// Mitsubishi GX Works2 project: 158-NGUYEN VAN CU   PLC: FX3G

PROGRAM MAIN
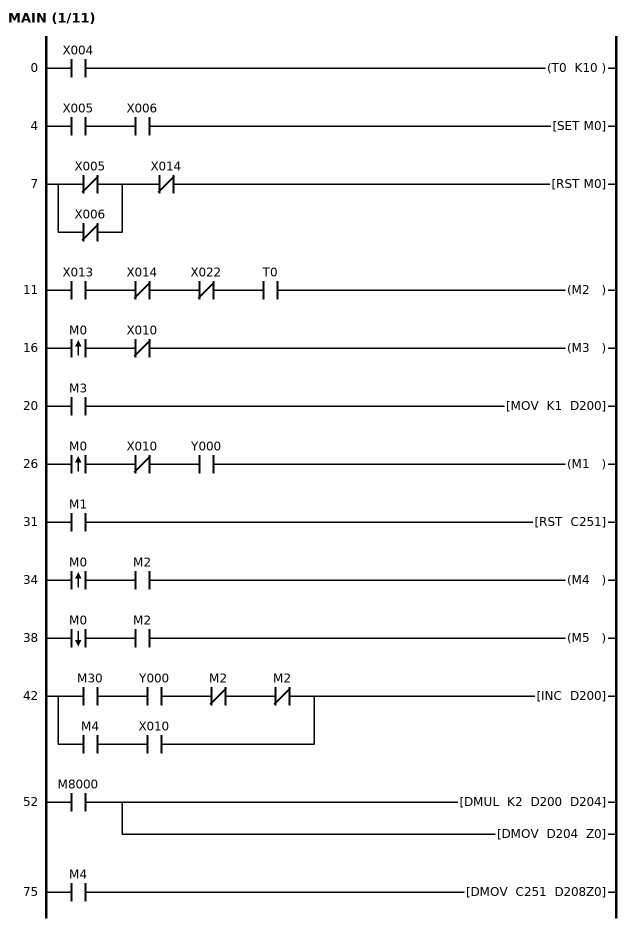
0     LD      X004
      OUT     T0 K10
4     LD      X005
      AND     X006
      SET     M0
7     LDI     X005
      ORI     X006
      ANI     X014
      RST     M0
11    LD      X013
      ANI     X014
      ANI     X022
      AND     T0
      OUT     M2
16    LDP     M0
      ANI     X010
      OUT     M3
20    LD      M3
      MOV     K1 D200
26    LDP     M0
      ANI     X010
      AND     Y000
      OUT     M1
31    LD      M1
      RST     C251
34    LDP     M0
      AND     M2
      OUT     M4
38    LDF     M0
      AND     M2
      OUT     M5
42    LD      M30
      AND     Y000
      ANI     M2
      ANI     M2
      LD      M4
      AND     X010
      ORB
      INC     D200
52    LD      M8000
      DMUL    K2 D200 D204
      DMOV    D204 Z0
75    LD      M4
      DMOV    C251 D208Z0
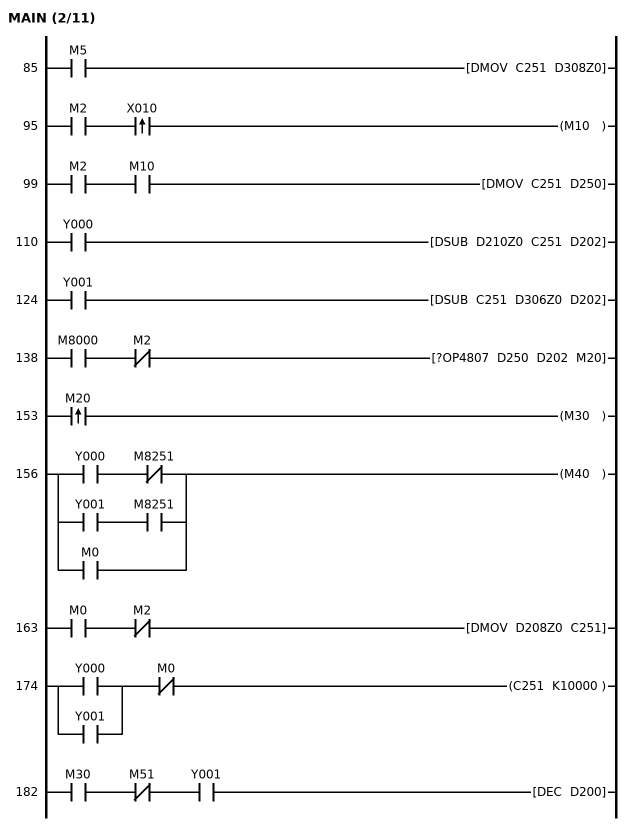
85    LD      M5
      DMOV    C251 D308Z0
95    LD      M2
      ANDP    X010
      OUT     M10
99    LD      M2
      AND     M10
      DMOV    C251 D250
110   LD      Y000
      DSUB    D210Z0 C251 D202
124   LD      Y001
      DSUB    C251 D306Z0 D202
138   LD      M8000
      ANI     M2
      ?OP4807 D250 D202 M20
153   LDP     M20
      OUT     M30
156   LD      Y000
      ANI     M8251
      LD      Y001
      AND     M8251
      ORB
      OR      M0
      OUT     M40
163   LD      M0
      ANI     M2
      DMOV    D208Z0 C251
174   LD      Y000
      OR      Y001
      ANI     M0
      OUT     C251 K10000
182   LD      M30
      ANI     M51
      AND     Y001
      DEC     D200
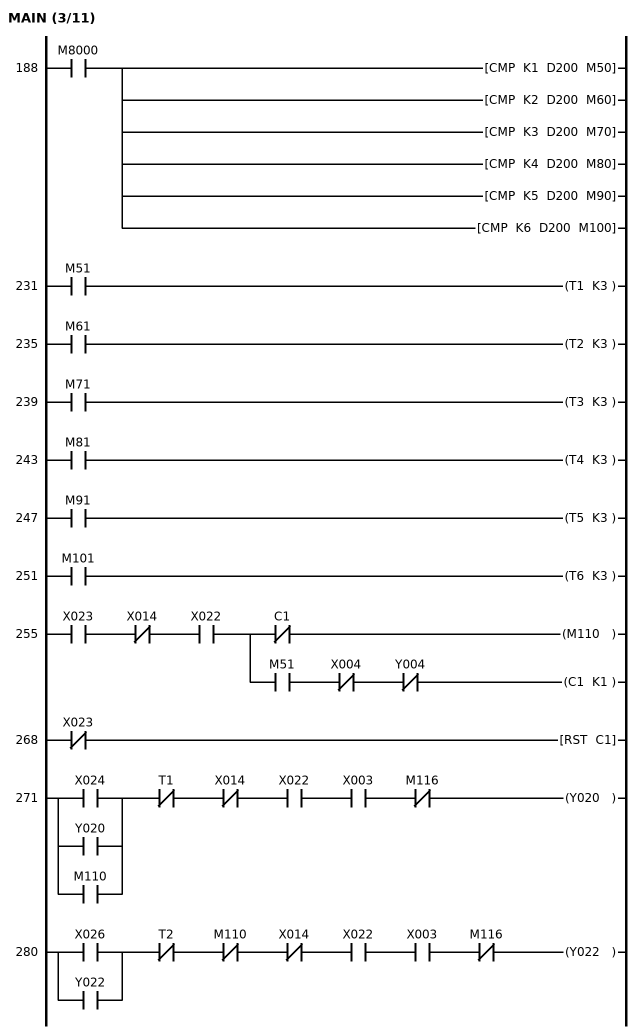
188   LD      M8000
      CMP     K1 D200 M50
      CMP     K2 D200 M60
      CMP     K3 D200 M70
      CMP     K4 D200 M80
      CMP     K5 D200 M90
      CMP     K6 D200 M100
231   LD      M51
      OUT     T1 K3
235   LD      M61
      OUT     T2 K3
239   LD      M71
      OUT     T3 K3
243   LD      M81
      OUT     T4 K3
247   LD      M91
      OUT     T5 K3
251   LD      M101
      OUT     T6 K3
255   LD      X023
      ANI     X014
      AND     X022
      MPS
      ANI     C1
      OUT     M110
      MPP
      AND     M51
      ANI     X004
      ANI     Y004
      OUT     C1 K1
268   LDI     X023
      RST     C1
271   LD      X024
      OR      Y020
      OR      M110
      ANI     T1
      ANI     X014
      AND     X022
      AND     X003
      ANI     M116
      OUT     Y020
280   LD      X026
      OR      Y022
      ANI     T2
      ANI     M110
      ANI     X014
      AND     X022
      AND     X003
      ANI     M116
      OUT     Y022
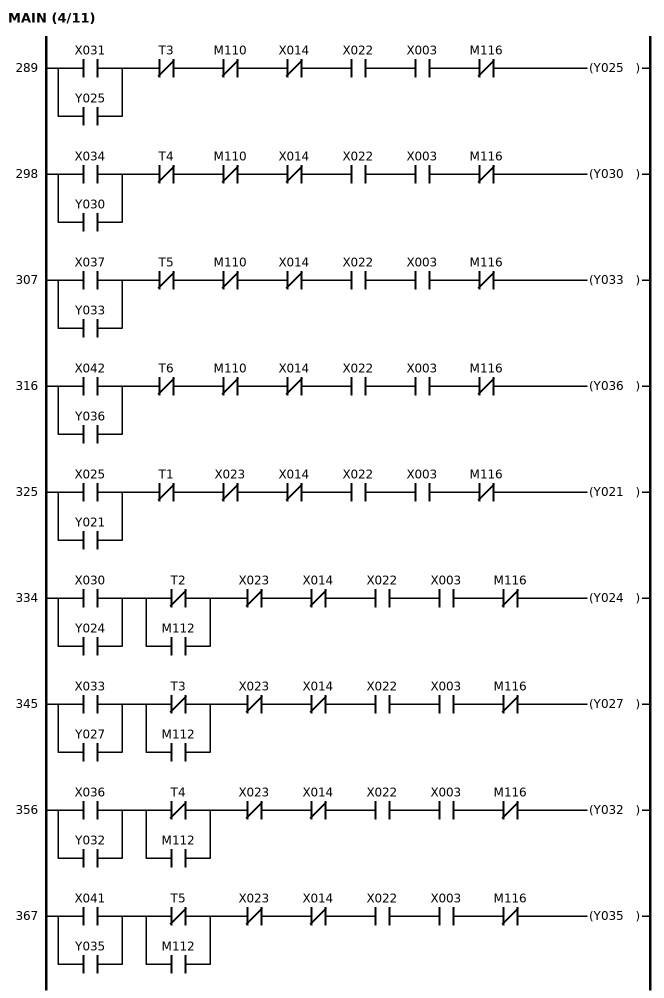
289   LD      X031
      OR      Y025
      ANI     T3
      ANI     M110
      ANI     X014
      AND     X022
      AND     X003
      ANI     M116
      OUT     Y025
298   LD      X034
      OR      Y030
      ANI     T4
      ANI     M110
      ANI     X014
      AND     X022
      AND     X003
      ANI     M116
      OUT     Y030
307   LD      X037
      OR      Y033
      ANI     T5
      ANI     M110
      ANI     X014
      AND     X022
      AND     X003
      ANI     M116
      OUT     Y033
316   LD      X042
      OR      Y036
      ANI     T6
      ANI     M110
      ANI     X014
      AND     X022
      AND     X003
      ANI     M116
      OUT     Y036
325   LD      X025
      OR      Y021
      ANI     T1
      ANI     X023
      ANI     X014
      AND     X022
      AND     X003
      ANI     M116
      OUT     Y021
334   LD      X030
      OR      Y024
      LDI     T2
      OR      M112
      ANB
      ANI     X023
      ANI     X014
      AND     X022
      AND     X003
      ANI     M116
      OUT     Y024
345   LD      X033
      OR      Y027
      LDI     T3
      OR      M112
      ANB
      ANI     X023
      ANI     X014
      AND     X022
      AND     X003
      ANI     M116
      OUT     Y027
356   LD      X036
      OR      Y032
      LDI     T4
      OR      M112
      ANB
      ANI     X023
      ANI     X014
      AND     X022
      AND     X003
      ANI     M116
      OUT     Y032
367   LD      X041
      OR      Y035
      LDI     T5
      OR      M112
      ANB
      ANI     X023
      ANI     X014
      AND     X022
      AND     X003
      ANI     M116
      OUT     Y035
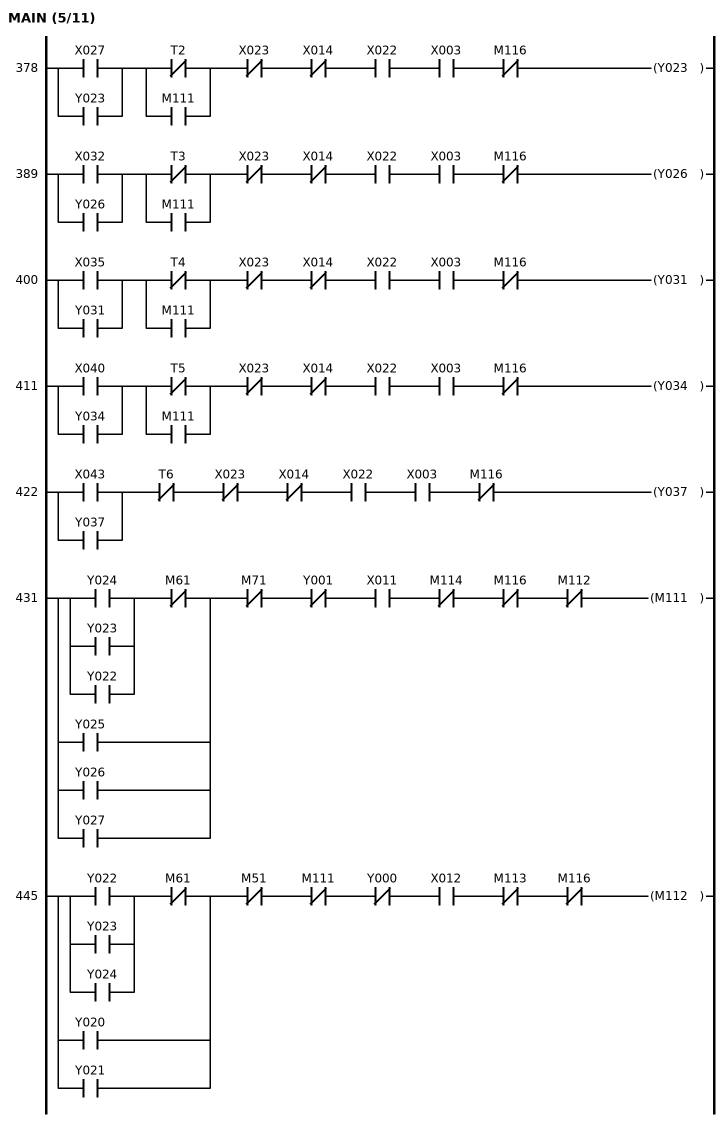
378   LD      X027
      OR      Y023
      LDI     T2
      OR      M111
      ANB
      ANI     X023
      ANI     X014
      AND     X022
      AND     X003
      ANI     M116
      OUT     Y023
389   LD      X032
      OR      Y026
      LDI     T3
      OR      M111
      ANB
      ANI     X023
      ANI     X014
      AND     X022
      AND     X003
      ANI     M116
      OUT     Y026
400   LD      X035
      OR      Y031
      LDI     T4
      OR      M111
      ANB
      ANI     X023
      ANI     X014
      AND     X022
      AND     X003
      ANI     M116
      OUT     Y031
411   LD      X040
      OR      Y034
      LDI     T5
      OR      M111
      ANB
      ANI     X023
      ANI     X014
      AND     X022
      AND     X003
      ANI     M116
      OUT     Y034
422   LD      X043
      OR      Y037
      ANI     T6
      ANI     X023
      ANI     X014
      AND     X022
      AND     X003
      ANI     M116
      OUT     Y037
431   LD      Y024
      OR      Y023
      OR      Y022
      ANI     M61
      OR      Y025
      OR      Y026
      OR      Y027
      ANI     M71
      ANI     Y001
      AND     X011
      ANI     M114
      ANI     M116
      ANI     M112
      OUT     M111
445   LD      Y022
      OR      Y023
      OR      Y024
      ANI     M61
      OR      Y020
      OR      Y021
      ANI     M51
      ANI     M111
      ANI     Y000
      AND     X012
      ANI     M113
      ANI     M116
      OUT     M112
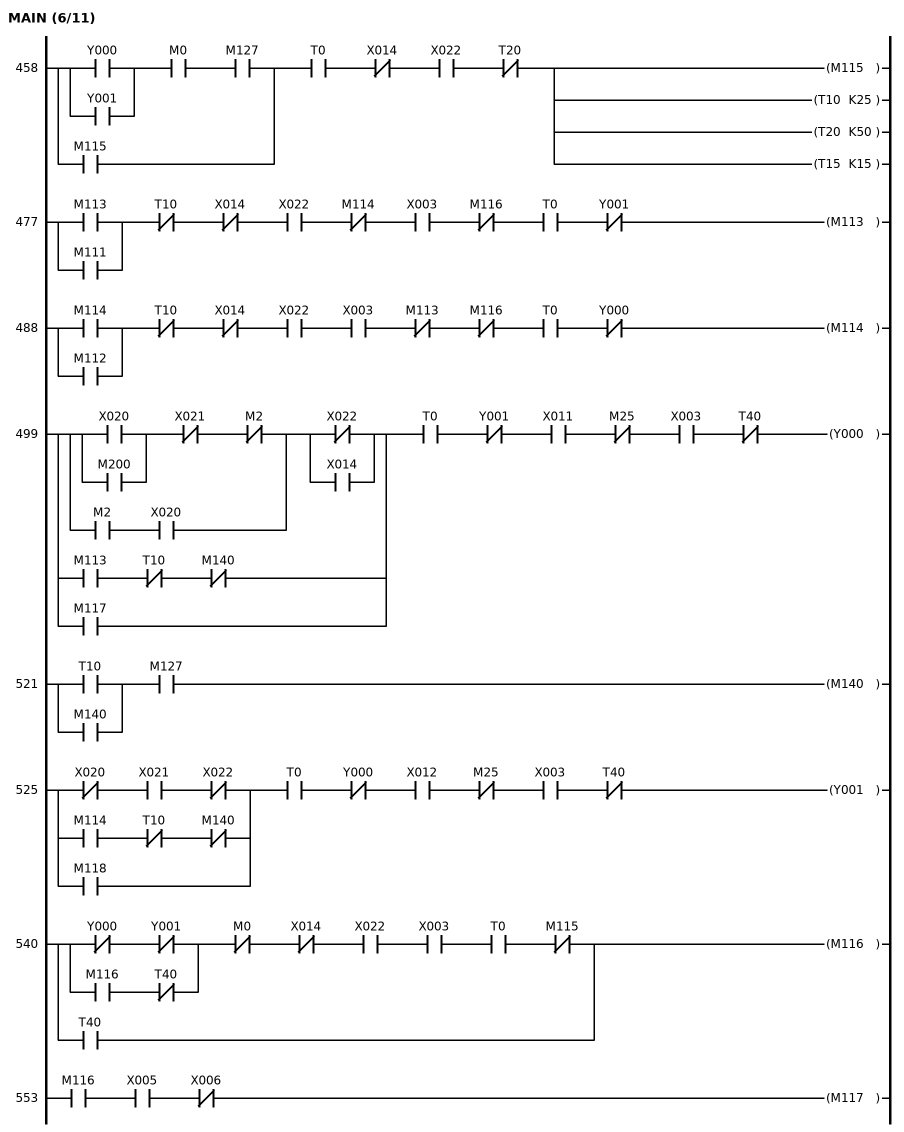
458   LD      Y000
      OR      Y001
      AND     M0
      AND     M127
      OR      M115
      AND     T0
      ANI     X014
      AND     X022
      ANI     T20
      OUT     M115
      OUT     T10 K25
      OUT     T20 K50
      OUT     T15 K15
477   LD      M113
      OR      M111
      ANI     T10
      ANI     X014
      AND     X022
      ANI     M114
      AND     X003
      ANI     M116
      AND     T0
      ANI     Y001
      OUT     M113
488   LD      M114
      OR      M112
      ANI     T10
      ANI     X014
      AND     X022
      AND     X003
      ANI     M113
      ANI     M116
      AND     T0
      ANI     Y000
      OUT     M114
499   LD      X020
      OR      M200
      ANI     X021
      ANI     M2
      LD      M2
      AND     X020
      ORB
      LDI     X022
      OR      X014
      ANB
      LD      M113
      ANI     T10
      ANI     M140
      ORB
      OR      M117
      AND     T0
      ANI     Y001
      AND     X011
      ANI     M25
      AND     X003
      ANI     T40
      OUT     Y000
521   LD      T10
      OR      M140
      AND     M127
      OUT     M140
525   LDI     X020
      AND     X021
      ANI     X022
      LD      M114
      ANI     T10
      ANI     M140
      ORB
      OR      M118
      AND     T0
      ANI     Y000
      AND     X012
      ANI     M25
      AND     X003
      ANI     T40
      OUT     Y001
540   LDI     Y000
      ANI     Y001
      LD      M116
      ANI     T40
      ORB
      ANI     M0
      ANI     X014
      AND     X022
      AND     X003
      AND     T0
      ANI     M115
      OR      T40
      OUT     M116
553   LD      M116
      AND     X005
      ANI     X006
      OUT     M117
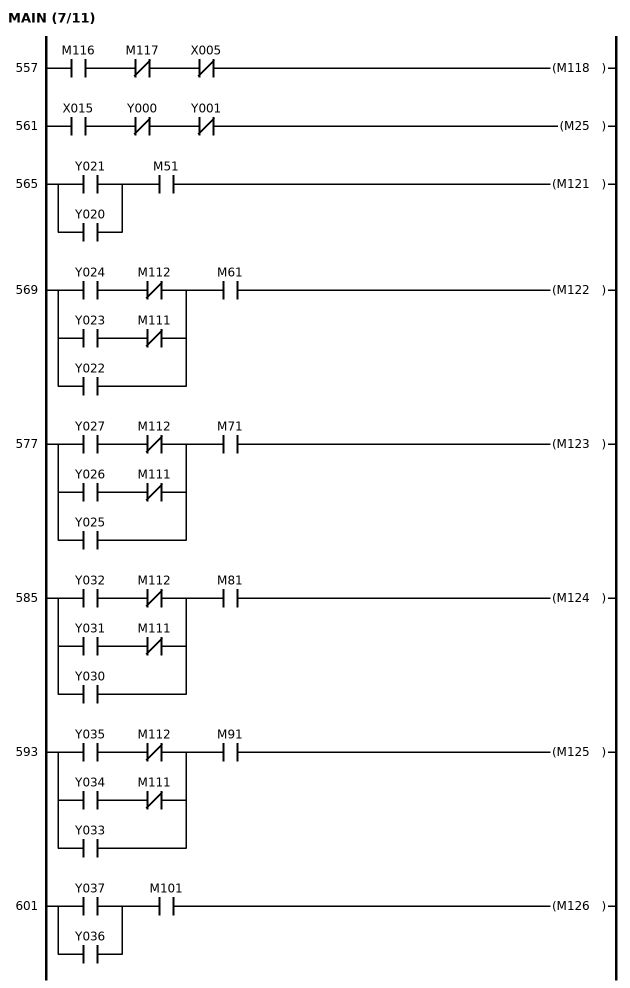
557   LD      M116
      ANI     M117
      ANI     X005
      OUT     M118
561   LD      X015
      ANI     Y000
      ANI     Y001
      OUT     M25
565   LD      Y021
      OR      Y020
      AND     M51
      OUT     M121
569   LD      Y024
      ANI     M112
      LD      Y023
      ANI     M111
      ORB
      OR      Y022
      AND     M61
      OUT     M122
577   LD      Y027
      ANI     M112
      LD      Y026
      ANI     M111
      ORB
      OR      Y025
      AND     M71
      OUT     M123
585   LD      Y032
      ANI     M112
      LD      Y031
      ANI     M111
      ORB
      OR      Y030
      AND     M81
      OUT     M124
593   LD      Y035
      ANI     M112
      LD      Y034
      ANI     M111
      ORB
      OR      Y033
      AND     M91
      OUT     M125
601   LD      Y037
      OR      Y036
      AND     M101
      OUT     M126
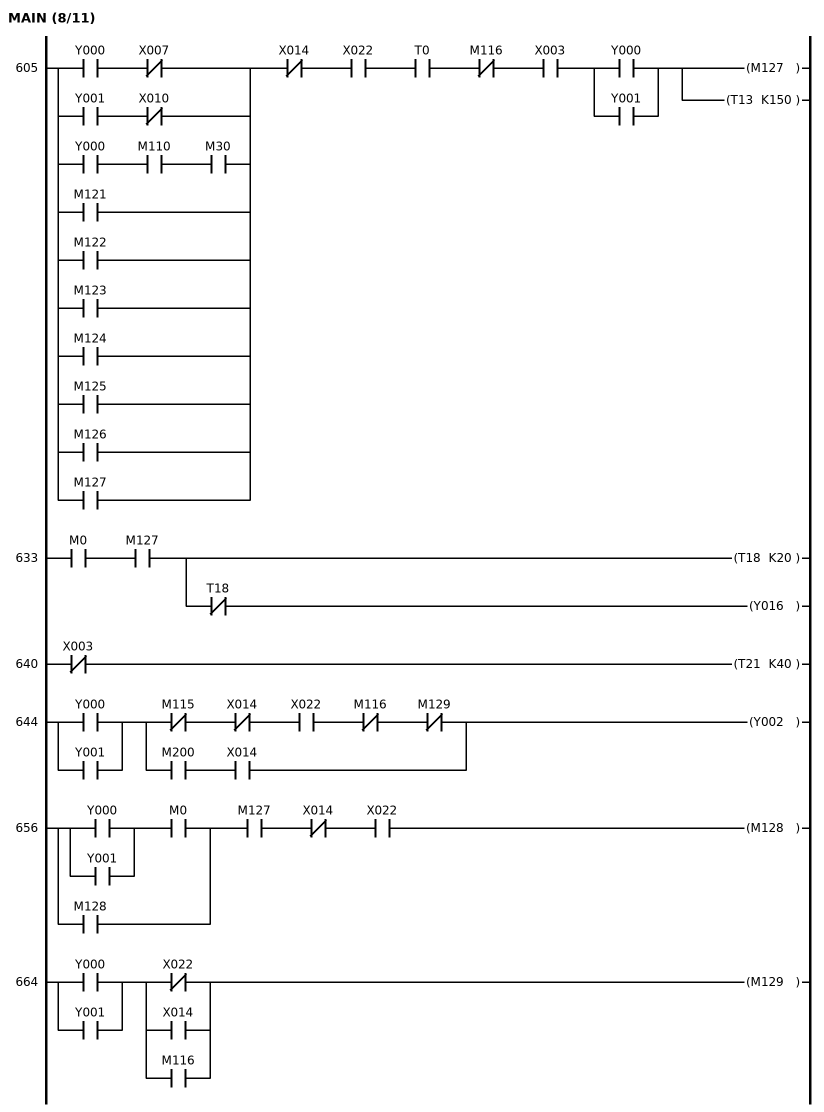
605   LD      Y000
      ANI     X007
      LD      Y001
      ANI     X010
      ORB
      LD      Y000
      AND     M110
      AND     M30
      ORB
      OR      M121
      OR      M122
      OR      M123
      OR      M124
      OR      M125
      OR      M126
      OR      M127
      ANI     X014
      AND     X022
      AND     T0
      ANI     M116
      AND     X003
      LD      Y000
      OR      Y001
      ANB
      OUT     M127
      OUT     T13 K150
633   LD      M0
      AND     M127
      OUT     T18 K20
      ANI     T18
      OUT     Y016
640   LDI     X003
      OUT     T21 K40
644   LD      Y000
      OR      Y001
      LDI     M115
      ANI     X014
      AND     X022
      ANI     M116
      ANI     M129
      LD      M200
      AND     X014
      ORB
      ANB
      OUT     Y002
656   LD      Y000
      OR      Y001
      AND     M0
      OR      M128
      AND     M127
      ANI     X014
      AND     X022
      OUT     M128
664   LD      Y000
      OR      Y001
      LDI     X022
      OR      X014
      OR      M116
      ANB
      OUT     M129
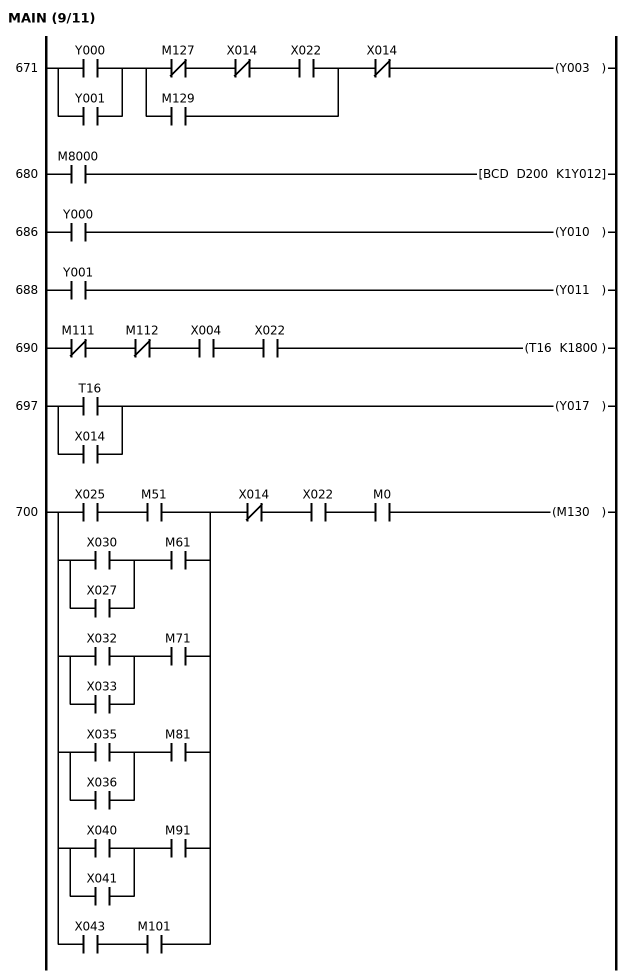
671   LD      Y000
      OR      Y001
      LDI     M127
      ANI     X014
      AND     X022
      OR      M129
      ANB
      ANI     X014
      OUT     Y003
680   LD      M8000
      BCD     D200 K1Y012
686   LD      Y000
      OUT     Y010
688   LD      Y001
      OUT     Y011
690   LDI     M111
      ANI     M112
      AND     X004
      AND     X022
      OUT     T16 K1800
697   LD      T16
      OR      X014
      OUT     Y017
700   LD      X025
      AND     M51
      LD      X030
      OR      X027
      AND     M61
      ORB
      LD      X032
      OR      X033
      AND     M71
      ORB
      LD      X035
      OR      X036
      AND     M81
      ORB
      LD      X040
      OR      X041
      AND     M91
      ORB
      LD      X043
      AND     M101
      ORB
      ANI     X014
      AND     X022
      AND     M0
      OUT     M130
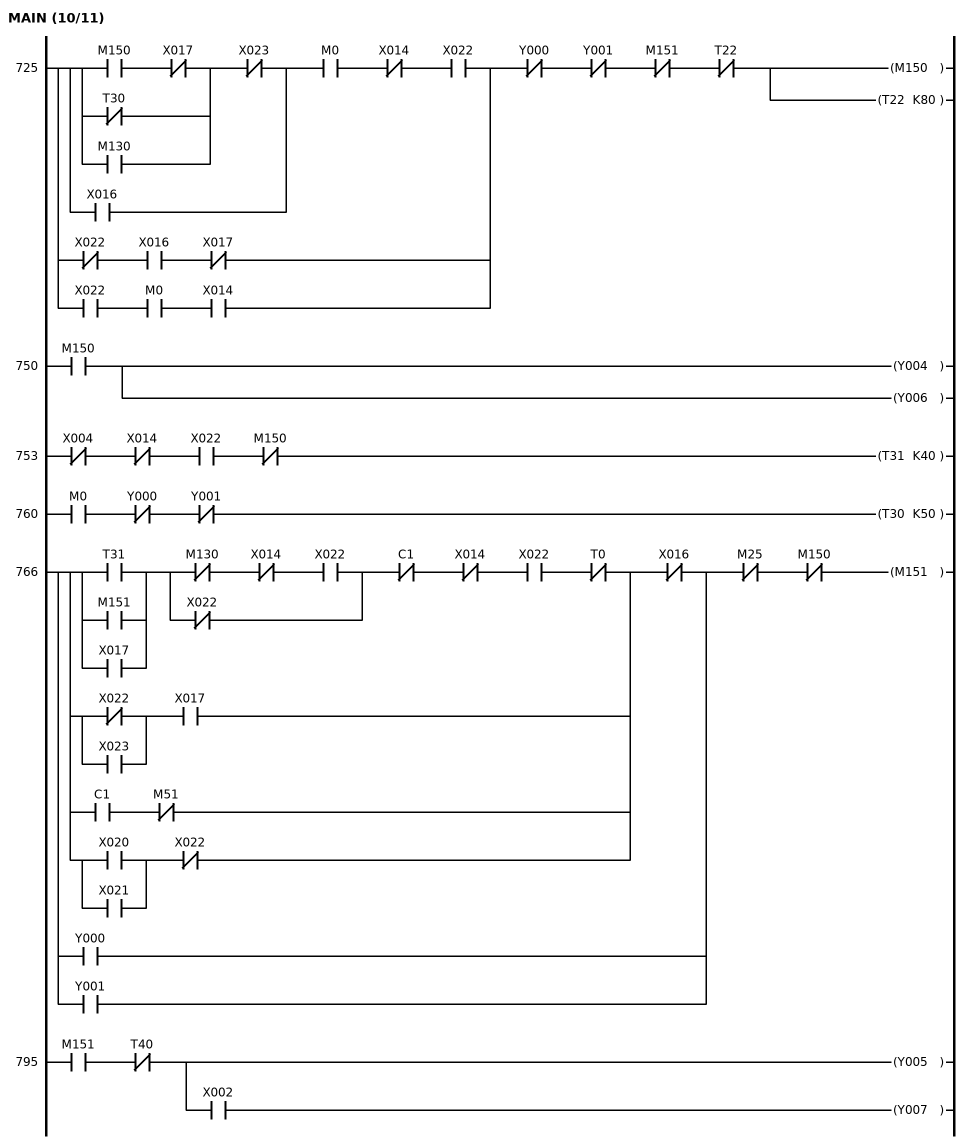
725   LD      M150
      ANI     X017
      ORI     T30
      OR      M130
      ANI     X023
      OR      X016
      AND     M0
      ANI     X014
      AND     X022
      LDI     X022
      AND     X016
      ANI     X017
      ORB
      LD      X022
      AND     M0
      AND     X014
      ORB
      ANI     Y000
      ANI     Y001
      ANI     M151
      ANI     T22
      OUT     M150
      OUT     T22 K80
750   LD      M150
      OUT     Y004
      OUT     Y006
753   LDI     X004
      ANI     X014
      AND     X022
      ANI     M150
      OUT     T31 K40
760   LD      M0
      ANI     Y000
      ANI     Y001
      OUT     T30 K50
766   LD      T31
      OR      M151
      OR      X017
      LDI     M130
      ANI     X014
      AND     X022
      ORI     X022
      ANB
      ANI     C1
      ANI     X014
      AND     X022
      ANI     T0
      LDI     X022
      OR      X023
      AND     X017
      ORB
      LD      C1
      ANI     M51
      ORB
      LD      X020
      OR      X021
      ANI     X022
      ORB
      ANI     X016
      OR      Y000
      OR      Y001
      ANI     M25
      ANI     M150
      OUT     M151
795   LD      M151
      ANI     T40
      OUT     Y005
      AND     X002
      OUT     Y007
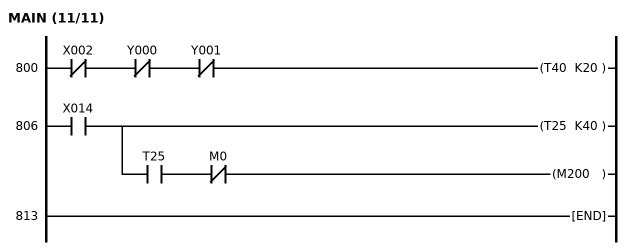
800   LDI     X002
      ANI     Y000
      ANI     Y001
      OUT     T40 K20
806   LD      X014
      OUT     T25 K40
      AND     T25
      ANI     M0
      OUT     M200
813   END
END_PROGRAM
